% RSLogix 500 project SOL2.RSS, saved by version 8.30.00.16 %
PROJECT "SOL2"    % processor: Bul.1763 MicroLogix 1100 Series B %

PROGRAM FILES
  LAD 2 "MAIN"  4 rungs
  LAD 3 "IO"  8 rungs
  LAD 4 "CONTROLS"  6 rungs
  LAD 5 "CYCLE"  5 rungs

DATA FILES
  O0 OUTPUT  4 elements
  I1 INPUT  6 elements
  S2 STATUS  66 elements
  B3 BINARY  1 elements
  T4 TIMER  1 elements
  C5 COUNTER  1 elements
  R6 CONTROL  1 elements
  N7 INTEGER  1 elements
  F8 FLOAT  1 elements

LADDER 2 "MAIN"
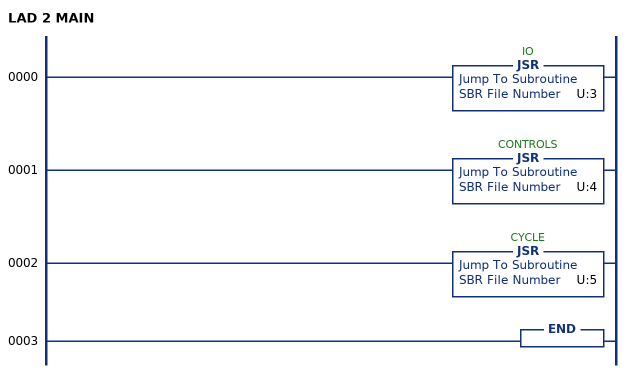
% Rung: 0 %
SOR JSR U:3 EOR
%   U:3  "IO" %
% Rung: 1 %
SOR JSR U:4 EOR
%   U:4  "CONTROLS" %
% Rung: 2 %
SOR JSR U:5 EOR
%   U:5  "CYCLE" %
% Rung: 3 %
SOR END EOR

LADDER 3 "IO"
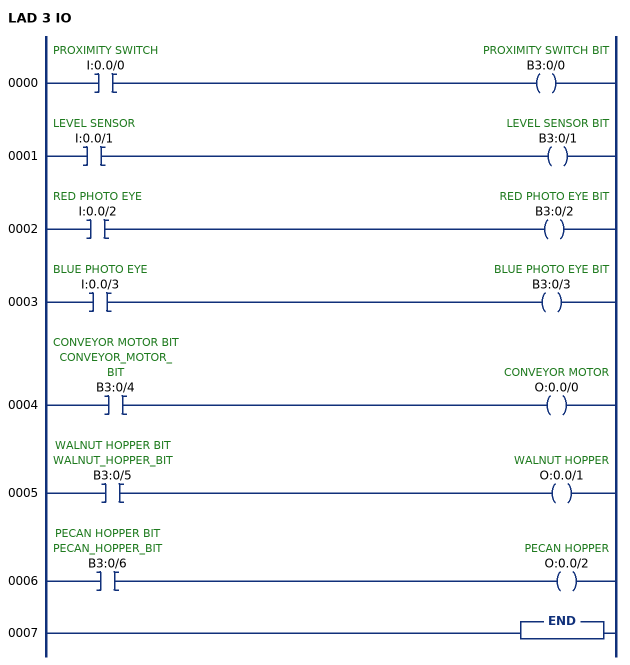
% Rung: 0 %
SOR XIC I:0.0/0 OTE B3:0/0 EOR
%   I:0.0/0  "PROXIMITY SWITCH" %
%   B3:0/0  "PROXIMITY SWITCH BIT" %
% Rung: 1 %
SOR XIC I:0.0/1 OTE B3:0/1 EOR
%   I:0.0/1  "LEVEL SENSOR" %
%   B3:0/1  "LEVEL SENSOR BIT" %
% Rung: 2 %
SOR XIC I:0.0/2 OTE B3:0/2 EOR
%   I:0.0/2  "RED PHOTO EYE" %
%   B3:0/2  "RED PHOTO EYE BIT" %
% Rung: 3 %
SOR XIC I:0.0/3 OTE B3:0/3 EOR
%   I:0.0/3  "BLUE PHOTO EYE" %
%   B3:0/3  "BLUE PHOTO EYE BIT" %
% Rung: 4 %
SOR XIC B3:0/4 OTE O:0.0/0 EOR
%   B3:0/4  CONVEYOR_MOTOR_BIT  "CONVEYOR MOTOR BIT" %
%   O:0.0/0  "CONVEYOR MOTOR" %
% Rung: 5 %
SOR XIC B3:0/5 OTE O:0.0/1 EOR
%   B3:0/5  WALNUT_HOPPER_BIT  "WALNUT HOPPER BIT" %
%   O:0.0/1  "WALNUT HOPPER" %
% Rung: 6 %
SOR XIC B3:0/6 OTE O:0.0/2 EOR
%   B3:0/6  PECAN_HOPPER_BIT  "PECAN HOPPER BIT" %
%   O:0.0/2  "PECAN HOPPER" %
% Rung: 7 %
SOR END EOR

LADDER 4 "CONTROLS"
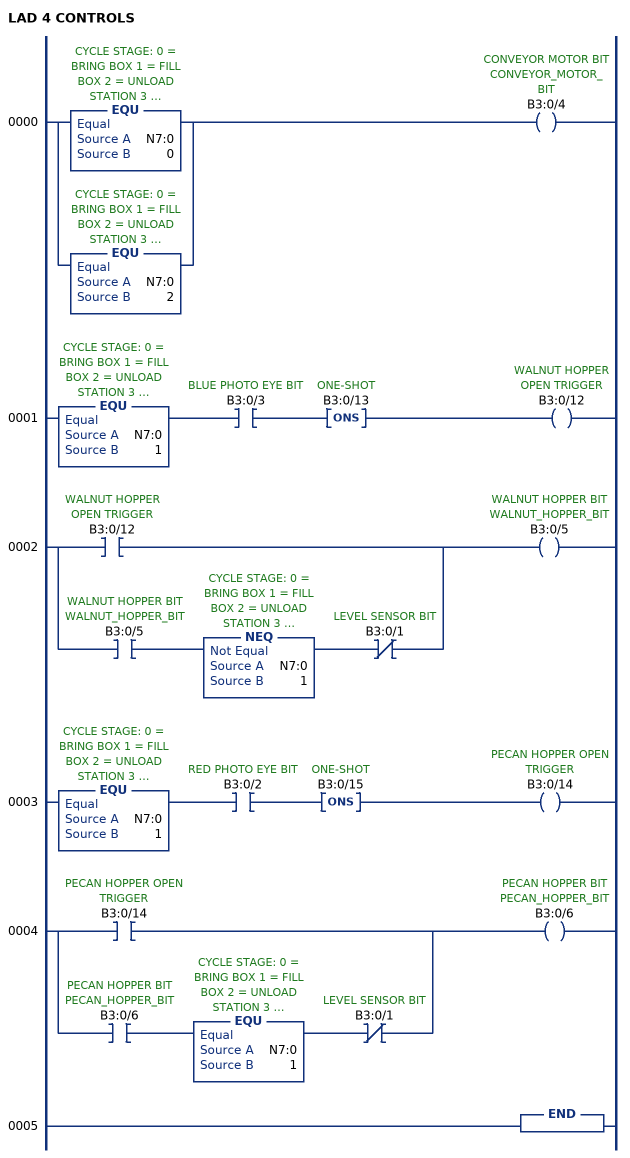
% Rung: 0 %
SOR BST EQU N7:0 0 NXB EQU N7:0 2 BND OTE B3:0/4 EOR
%   N7:0  "CYCLE STAGE: 0 = BRING BOX 1 = FILL BOX 2 = UNLOAD STATION 3 = INTERMEDIATE" %
%   B3:0/4  CONVEYOR_MOTOR_BIT  "CONVEYOR MOTOR BIT" %
% Rung: 1 %
SOR EQU N7:0 1 XIC B3:0/3 ONS B3:0/13 OTE B3:0/12 EOR
%   N7:0  "CYCLE STAGE: 0 = BRING BOX 1 = FILL BOX 2 = UNLOAD STATION 3 = INTERMEDIATE" %
%   B3:0/3  "BLUE PHOTO EYE BIT" %
%   B3:0/13  "ONE-SHOT" %
%   B3:0/12  "WALNUT HOPPER OPEN TRIGGER" %
% Rung: 2 %
SOR BST XIC B3:0/12 NXB XIC B3:0/5 NEQ N7:0 1 XIO B3:0/1 BND OTE B3:0/5 EOR
%   B3:0/12  "WALNUT HOPPER OPEN TRIGGER" %
%   B3:0/5  WALNUT_HOPPER_BIT  "WALNUT HOPPER BIT" %
%   N7:0  "CYCLE STAGE: 0 = BRING BOX 1 = FILL BOX 2 = UNLOAD STATION 3 = INTERMEDIATE" %
%   B3:0/1  "LEVEL SENSOR BIT" %
% Rung: 3 %
SOR EQU N7:0 1 XIC B3:0/2 ONS B3:0/15 OTE B3:0/14 EOR
%   N7:0  "CYCLE STAGE: 0 = BRING BOX 1 = FILL BOX 2 = UNLOAD STATION 3 = INTERMEDIATE" %
%   B3:0/2  "RED PHOTO EYE BIT" %
%   B3:0/15  "ONE-SHOT" %
%   B3:0/14  "PECAN HOPPER OPEN TRIGGER" %
% Rung: 4 %
SOR BST XIC B3:0/14 NXB XIC B3:0/6 EQU N7:0 1 XIO B3:0/1 BND OTE B3:0/6 EOR
%   B3:0/14  "PECAN HOPPER OPEN TRIGGER" %
%   B3:0/6  PECAN_HOPPER_BIT  "PECAN HOPPER BIT" %
%   N7:0  "CYCLE STAGE: 0 = BRING BOX 1 = FILL BOX 2 = UNLOAD STATION 3 = INTERMEDIATE" %
%   B3:0/1  "LEVEL SENSOR BIT" %
% Rung: 5 %
SOR END EOR

LADDER 5 "CYCLE"
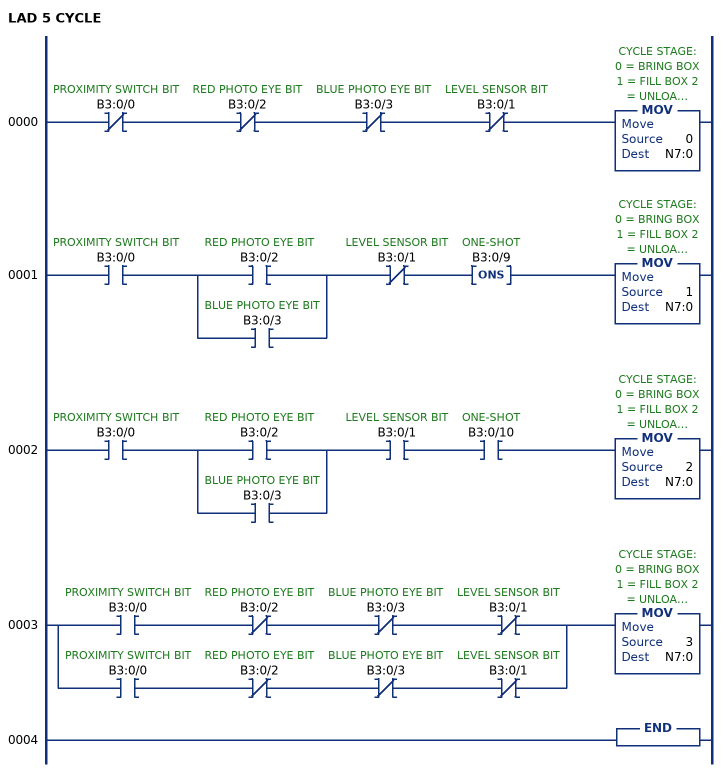
% Rung: 0 %
SOR XIO B3:0/0 XIO B3:0/2 XIO B3:0/3 XIO B3:0/1 MOV 0 N7:0 EOR
%   B3:0/0  "PROXIMITY SWITCH BIT" %
%   B3:0/2  "RED PHOTO EYE BIT" %
%   B3:0/3  "BLUE PHOTO EYE BIT" %
%   B3:0/1  "LEVEL SENSOR BIT" %
%   N7:0  "CYCLE STAGE: 0 = BRING BOX 1 = FILL BOX 2 = UNLOAD STATION 3 = INTERMEDIATE" %
% Rung: 1 %
SOR XIC B3:0/0 BST XIC B3:0/2 NXB XIC B3:0/3 BND XIO B3:0/1 ONS B3:0/9 MOV 1 N7:0 EOR
%   B3:0/0  "PROXIMITY SWITCH BIT" %
%   B3:0/2  "RED PHOTO EYE BIT" %
%   B3:0/3  "BLUE PHOTO EYE BIT" %
%   B3:0/1  "LEVEL SENSOR BIT" %
%   B3:0/9  "ONE-SHOT" %
%   N7:0  "CYCLE STAGE: 0 = BRING BOX 1 = FILL BOX 2 = UNLOAD STATION 3 = INTERMEDIATE" %
% Rung: 2 %
SOR XIC B3:0/0 BST XIC B3:0/2 NXB XIC B3:0/3 BND XIC B3:0/1 XIC B3:0/10 MOV 2 N7:0 EOR
%   B3:0/0  "PROXIMITY SWITCH BIT" %
%   B3:0/2  "RED PHOTO EYE BIT" %
%   B3:0/3  "BLUE PHOTO EYE BIT" %
%   B3:0/1  "LEVEL SENSOR BIT" %
%   B3:0/10  "ONE-SHOT" %
%   N7:0  "CYCLE STAGE: 0 = BRING BOX 1 = FILL BOX 2 = UNLOAD STATION 3 = INTERMEDIATE" %
% Rung: 3 %
SOR BST XIC B3:0/0 XIO B3:0/2 XIO B3:0/3 XIO B3:0/1 NXB XIC B3:0/0 XIO B3:0/2 XIO B3:0/3 XIO B3:0/1 BND MOV 3 N7:0 EOR
%   B3:0/0  "PROXIMITY SWITCH BIT" %
%   B3:0/2  "RED PHOTO EYE BIT" %
%   B3:0/3  "BLUE PHOTO EYE BIT" %
%   B3:0/1  "LEVEL SENSOR BIT" %
%   N7:0  "CYCLE STAGE: 0 = BRING BOX 1 = FILL BOX 2 = UNLOAD STATION 3 = INTERMEDIATE" %
% Rung: 4 %
SOR END EOR

OTHER DOCUMENTED ADDRESSES
  B3:0/7  "CONVERYOR MOTOR START BIT"
  B3:0/8  "CONVEYOR MOTOR INTERRUPT"
  B3:0/11  "ONE-SHOT"
